TYPE StatsFailure :
STRUCT
	TimeStamp: TimeStamp;
	StationID: DINT;
	FailureID: DINT;
	Parameters: STRING;
END_STRUCT
END_TYPE

(* stored: Version 1.1.0.1, ProductVersion 3.1.4024.9
   DUT StatsFailure: Id {b0bded46-b8be-4ea0-bc58-a0af8295d0b4} *)
